(* PLC project PlcMain, Beckhoff Automation GmbH TwinCAT PLC Control 3.5.13.21 *)
(* stored: creationDateTime 2022-08-19T12:33:57.5074085, modificationDateTime 2022-08-19T12:33:57.5074085 *)

{attribute 'qualified_only'}
{attribute 'strict'}
TYPE StateDisp :
(
	Off := 0,
	Reset,
	PowerUp,
	Idle,
	Dispensing,
	Done
);
END_TYPE
